FUNCTION_BLOCK FB_Janitza
VAR_IN_OUT
	get					: ST_PowerMonitor_get;
	b_ThirdOutputFieldAvailable	: BOOL;
	b_NeutralTransformerAvailable: BOOL;
	b_InputFieldsAvailable		: BOOL;
END_VAR
VAR
	MBRead: FB_MBReadRegs;
	t_MBTimeout				: 	TIME := T#500MS;
	w_MBStartAddress		:	WORD;
	//Set 1 is bigger, as this includes voltage measurements.
	DataBuffer				: 	ARRAY[0..62] OF REAL;
	//SecondDataBuffer		: 	ARRAY[0..62] OF REAL;
	UI_Iterator	:	UINT;
	//retrieve new data every 100ms
	GetDataTimer	:	TON := (PT := TIME#50MS);
	
	di_RotationState		: DINT;
	
	ton_DelaySFCTip			: TON := (PT := T#10MS);
	
	
END_VAR

VAR_INPUT
	ReadData: BOOL;
	b_TNmodeEnable		AT %Q* : BOOL;
	
END_VAR

VAR
	ast_InputPowerlockData	:	ARRAY[1..2] OF ST_MeasurementFieldData;
	ast_OutputPowerlockData	:	ARRAY[1..3] OF ST_MeasurementFieldData;

	StartTransmissionEdge : R_Trig;
	TransmissionDone	:	F_trig;
	
	ui_MBRetryCount	:	uint;
	
	b_busy: BOOL;
	b_CommError: BOOL;
	udi_errid: UDINT;
	udi_cbread: UDINT;
	
END_VAR

//Initialization
get.events.b_MBCommWarning := FALSE;
get.events.b_MBCommError := FALSE;

MBread(tTimeOut := t_MBTimeout);

//While ReadData is true, initiate data transfer every 100ms;
GetDataTimer(in:= ((NOT GetDataTimer.Q) AND ReadData));

//ReadJanitzaData();
ReadDataSFC();

ACTION aCombineInputData:
IF b_InputFieldsAvailable THEN
	//Combine shared data from output fields into get struct
	get.InputField.ar_Current[Phases.L1] :=	get.InputField.powerlock[1].ar_Current[Phases.L1] + 
											get.InputField.Powerlock[2].ar_Current[Phases.L1];
	
	get.InputField.ar_Current[Phases.L2] :=	get.InputField.powerlock[1].ar_Current[Phases.L2] + 
											get.InputField.powerlock[2].ar_Current[Phases.L2];
	
	get.InputField.ar_Current[Phases.L3] :=	get.InputField.powerlock[1].ar_Current[Phases.L3] + 
											get.InputField.powerlock[2].ar_Current[Phases.L3];			
	
	get.InputField.ar_Current[Phases.N] :=	get.InputField.powerlock[1].ar_Current[Phases.N] + 
											get.InputField.powerlock[2].ar_Current[Phases.N];			
	
	get.InputField.ar_Current[Phases.AVG] :=	(get.InputField.ar_Current[Phases.L1] + 
											get.InputField.ar_Current[Phases.L2] +
											get.InputField.ar_Current[Phases.L3])/3;							
	
	Get.InputField.ar_ActivePower[Phases.L1]	:=	get.InputField.powerlock[1].ar_ActivePower[Phases.L1] + get.InputField.powerlock[2].ar_ActivePower[Phases.L1];
	Get.InputField.ar_ActivePower[Phases.L2]	:=	get.InputField.powerlock[1].ar_ActivePower[Phases.L2] + get.InputField.powerlock[2].ar_ActivePower[Phases.L2];
	Get.InputField.ar_ActivePower[Phases.L3]	:=	get.InputField.powerlock[1].ar_ActivePower[Phases.L3] + get.InputField.powerlock[2].ar_ActivePower[Phases.L3];
	Get.InputField.ar_ActivePower[Phases.AVG]	:=	get.InputField.powerlock[1].ar_ActivePower[Phases.AVG] + get.InputField.powerlock[2].ar_ActivePower[Phases.AVG];									
	Get.InputField.ar_ApparentPower[Phases.L1]	:=	get.InputField.powerlock[1].ar_ApparentPower[Phases.L1] + get.InputField.powerlock[2].ar_ApparentPower[Phases.L1];
	Get.InputField.ar_ApparentPower[Phases.L2]	:=	get.InputField.powerlock[1].ar_ApparentPower[Phases.L2] + get.InputField.powerlock[2].ar_ApparentPower[Phases.L2];	
	Get.InputField.ar_ApparentPower[Phases.L3]	:=	get.InputField.powerlock[1].ar_ApparentPower[Phases.L3] + get.InputField.powerlock[2].ar_ApparentPower[Phases.L3];
	Get.InputField.ar_ApparentPower[Phases.AVG]	:=	get.InputField.powerlock[1].ar_ApparentPower[Phases.AVG] + get.InputField.powerlock[2].ar_ApparentPower[Phases.AVG];												
	Get.InputField.ar_ReactivePower[Phases.L1]	:=	get.InputField.powerlock[1].ar_ReactivePower[Phases.L1] + get.InputField.powerlock[2].ar_ReactivePower[Phases.L1];
	Get.InputField.ar_ReactivePower[Phases.L2]	:=	get.InputField.powerlock[1].ar_ReactivePower[Phases.L2] + get.InputField.powerlock[2].ar_ReactivePower[Phases.L2];											
	Get.InputField.ar_ReactivePower[Phases.L3]	:=	get.InputField.powerlock[1].ar_ReactivePower[Phases.L3] + get.InputField.powerlock[2].ar_ReactivePower[Phases.L3];								
	Get.InputField.ar_ReactivePower[Phases.AVG]	:=	get.InputField.powerlock[1].ar_ReactivePower[Phases.AVG] + get.InputField.powerlock[2].ar_ReactivePower[Phases.AVG];	

	Get.InputField.r_EnergyConsumed		:=	get.InputField.powerlock[1].r_EnergyConsumed + 
											get.InputField.powerlock[2].r_EnergyConsumed;
	
	Get.InputField.r_EnergySupplied		:=	get.InputField.powerlock[1].r_EnergySupplied + 
											get.InputField.powerlock[2].r_EnergySupplied;
	
	get.InputField.ar_PowerFactor[Phases.L1] 	:=  PowerFactor(Get.InputField.ar_activePower[Phases.L1], Get.InputField.ar_ApparentPower[Phases.L1], Get.InputField.ar_ReactivePower[Phases.L1]); 										
	get.InputField.ar_PowerFactor[Phases.L2] 	:=  PowerFactor(Get.InputField.ar_activePower[Phases.L2], Get.InputField.ar_ApparentPower[Phases.L2], Get.InputField.ar_ReactivePower[Phases.L2]); 		
	get.InputField.ar_PowerFactor[Phases.L3] 	:=  PowerFactor(Get.InputField.ar_activePower[Phases.L3], Get.InputField.ar_ApparentPower[Phases.L3], Get.InputField.ar_ReactivePower[Phases.L3]); 									
	get.InputField.ar_THD[Phases.L1] 		:=		(ast_InputPowerLockData[1].ar_THD[Phases.L1] + ast_InputPowerLockData[2].ar_THD[Phases.L1])/2;		
	get.InputField.ar_THD[Phases.L2] 		:=		(ast_InputPowerLockData[1].ar_THD[Phases.L2] + ast_InputPowerLockData[2].ar_THD[Phases.L2])/2;	
	get.InputField.ar_THD[Phases.L3]		:=		(ast_InputPowerLockData[1].ar_THD[Phases.L3] + ast_InputPowerLockData[2].ar_THD[Phases.L3])/2;											
	get.InputField.ar_PowerFactor[Phases.AVG] :=	(get.InputField.ar_PowerFactor[Phases.L1] + get.InputField.ar_PowerFactor[Phases.L2] + get.InputField.ar_PowerFactor[Phases.L3])/3;		
	get.InputField.ar_THD[Phases.AVG] :=			(get.InputField.ar_THD[Phases.L1] + get.InputField.ar_THD[Phases.L2] + get.InputField.ar_THD[Phases.L3])/3;
END_IF
END_ACTION

ACTION aCombineOutputData:
//Combine shared data from output fields into get struct
get.OutputField.ar_Current[Phases.L1] 	:=	get.OutputField.powerlock[1].ar_current[Phases.L1] + get.OutputField.powerlock[2].ar_current[Phases.L1] + get.OutputField.powerlock[3].ar_current[Phases.L1];
get.OutputField.ar_Current[Phases.L2] 	:=	get.OutputField.powerlock[1].ar_current[Phases.L2] + get.OutputField.powerlock[2].ar_current[Phases.L2] + get.OutputField.powerlock[3].ar_current[Phases.L2];
get.OutputField.ar_Current[Phases.L3] 	:=	get.OutputField.powerlock[1].ar_current[Phases.L3] + get.OutputField.powerlock[2].ar_current[Phases.L3] + get.OutputField.powerlock[3].ar_current[Phases.L3];			
get.OutputField.ar_Current[Phases.N] 	:=	get.OutputField.powerlock[1].ar_current[Phases.N] + get.OutputField.powerlock[2].ar_current[Phases.N] + get.OutputField.powerlock[3].ar_current[Phases.N];			
get.OutputField.ar_Current[Phases.AVG] :=	(get.OutputField.ar_Current[Phases.L1] + get.OutputField.ar_Current[Phases.L2] + get.OutputField.ar_Current[Phases.L3])/3;							

Get.OutputField.ar_ActivePower[Phases.L1]		:=	get.outputfield.powerlock[1].ar_ActivePower[Phases.L1] + 
													get.outputfield.powerlock[2].ar_ActivePower[Phases.L1] +
													get.outputfield.powerlock[3].ar_ActivePower[Phases.L1];
Get.OutputField.ar_ActivePower[Phases.L2]		:=	get.outputfield.powerlock[1].ar_ActivePower[Phases.L2] + 
													get.outputfield.powerlock[2].ar_ActivePower[Phases.L2] +
													get.outputfield.powerlock[3].ar_ActivePower[Phases.L2];				
Get.OutputField.ar_ActivePower[Phases.L3]		:=	get.outputfield.powerlock[1].ar_ActivePower[Phases.L3] + 
													get.outputfield.powerlock[2].ar_ActivePower[Phases.L3] + 
													get.outputfield.powerlock[3].ar_ActivePower[Phases.L3];												
Get.OutputField.ar_ActivePower[Phases.AVG]		:=	get.outputfield.powerlock[1].ar_ActivePower[Phases.AVG] + 
													get.outputfield.powerlock[2].ar_ActivePower[Phases.AVG] +
													get.outputfield.powerlock[3].ar_ActivePower[Phases.AVG];																				
Get.OutputField.ar_ApparentPower[Phases.L1]		:=	get.outputfield.powerlock[1].ar_ApparentPower[Phases.L1] + 
													get.outputfield.powerlock[2].ar_ApparentPower[Phases.L1] +
													get.outputfield.powerlock[3].ar_ApparentPower[Phases.L1];
Get.OutputField.ar_ApparentPower[Phases.L2]		:=	get.outputfield.powerlock[1].ar_ApparentPower[Phases.L2] + 
													get.outputfield.powerlock[2].ar_ApparentPower[Phases.L2] +
													get.outputfield.powerlock[3].ar_ApparentPower[Phases.L2];													
Get.OutputField.ar_ApparentPower[Phases.L3]		:=	get.outputfield.powerlock[1].ar_ApparentPower[Phases.L3] + 
													get.outputfield.powerlock[2].ar_ApparentPower[Phases.L3] +
													get.outputfield.powerlock[3].ar_ApparentPower[Phases.L3];													
Get.OutputField.ar_ApparentPower[Phases.AVG]	:=	get.outputfield.powerlock[1].ar_ApparentPower[Phases.AVG] + 
													get.outputfield.powerlock[2].ar_ApparentPower[Phases.AVG] +
													get.outputfield.powerlock[3].ar_ApparentPower[Phases.AVG];																																								
Get.OutputField.ar_ReactivePower[Phases.L1]		:=	get.outputfield.powerlock[1].ar_ReactivePower[Phases.L1] + 
													get.outputfield.powerlock[2].ar_ReactivePower[Phases.L1] +
													get.outputfield.powerlock[3].ar_ReactivePower[Phases.L1];		
Get.OutputField.ar_ReactivePower[Phases.L2]		:=	get.outputfield.powerlock[1].ar_ReactivePower[Phases.L2] + 
													get.outputfield.powerlock[2].ar_ReactivePower[Phases.L2] +
													get.outputfield.powerlock[3].ar_ReactivePower[Phases.L2];															
Get.OutputField.ar_ReactivePower[Phases.L3]		:=	get.outputfield.powerlock[1].ar_ReactivePower[Phases.L3] + 
													get.outputfield.powerlock[2].ar_ReactivePower[Phases.L3] +
													get.outputfield.powerlock[3].ar_ReactivePower[Phases.L3];															
Get.OutputField.ar_ReactivePower[Phases.AVG]	:=	get.outputfield.powerlock[1].ar_ReactivePower[Phases.AVG] + 
													get.outputfield.powerlock[2].ar_ReactivePower[Phases.AVG] +	
													get.outputfield.powerlock[3].ar_ReactivePower[Phases.AVG];																					
Get.OutputField.r_EnergyConsumed				:=	get.outputfield.powerlock[1].r_EnergyConsumed + 
													get.outputfield.powerlock[2].r_EnergyConsumed + 
													get.outputfield.powerlock[3].r_EnergyConsumed;
Get.OutputField.r_EnergySupplied				:=	get.outputfield.powerlock[1].r_EnergySupplied + 
													get.outputfield.powerlock[2].r_EnergySupplied + 
													get.outputfield.powerlock[3].r_EnergySupplied;
get.OutputField.ar_PowerFactor[Phases.L1] 		:=  PowerFactor(Get.OutputField.ar_activePower[Phases.L1], Get.OutputField.ar_ApparentPower[Phases.L1], Get.OutputField.ar_ReactivePower[Phases.L1]); 										
get.OutputField.ar_PowerFactor[Phases.L2] 		:=  PowerFactor(Get.OutputField.ar_activePower[Phases.L2], Get.OutputField.ar_ApparentPower[Phases.L2], Get.OutputField.ar_ReactivePower[Phases.L2]); 		
get.OutputField.ar_PowerFactor[Phases.L3] 		:=  PowerFactor(Get.OutputField.ar_activePower[Phases.L3], Get.OutputField.ar_ApparentPower[Phases.L3], Get.OutputField.ar_ReactivePower[Phases.L3]); 									

//if 3 output fields are available, calculate averages over 3 fields. Otherwise over 2
IF b_ThirdOutputFieldAvailable THEN
	get.OutputField.ar_THD[Phases.L1] 		:=	   (get.outputfield.powerlock[1].ar_THD[Phases.L1] + 
													get.outputfield.powerlock[2].ar_THD[Phases.L1] + 
													get.outputfield.powerlock[3].ar_THD[Phases.L1])/3;												
	get.OutputField.ar_THD[Phases.L2] 		:=     (get.outputfield.powerlock[1].ar_THD[Phases.L2] + 
													get.outputfield.powerlock[2].ar_THD[Phases.L2] + 
													get.outputfield.powerlock[3].ar_THD[Phases.L2])/3;		
	get.OutputField.ar_THD[Phases.L3]		 :=	   (get.outputfield.powerlock[1].ar_THD[Phases.L3] + 
													get.outputfield.powerlock[2].ar_THD[Phases.L3] + 
													get.outputfield.powerlock[3].ar_THD[Phases.L3])/3;														
ELSE
	get.OutputField.ar_THD[Phases.L1] 		:=	   (get.outputfield.powerlock[1].ar_THD[Phases.L1] + 
													get.outputfield.powerlock[2].ar_THD[Phases.L1])/2;											
	get.OutputField.ar_THD[Phases.L2] 		:=     (get.outputfield.powerlock[1].ar_THD[Phases.L2] + 
													get.outputfield.powerlock[2].ar_THD[Phases.L2])/2;	
	get.OutputField.ar_THD[Phases.L3]		 :=	   (get.outputfield.powerlock[1].ar_THD[Phases.L3] + 
													get.outputfield.powerlock[2].ar_THD[Phases.L3])/2;											
END_IF



get.OutputField.ar_PowerFactor[Phases.AVG] :=	(get.OutputField.ar_PowerFactor[Phases.L1] + 
												get.OutputField.ar_PowerFactor[Phases.L2] + 
												get.OutputField.ar_PowerFactor[Phases.L3])/3;		

get.OutputField.ar_THD[Phases.AVG] :=			(get.OutputField.ar_THD[Phases.L1] + 
												get.OutputField.ar_THD[Phases.L2] + 
												get.OutputField.ar_THD[Phases.L3])/3;
												
get.OutputField.r_VoltageUnbalance := 			LineUnbalance(
													r_L1 := get.OutputField.ar_LineVoltage[phases.L1],
													r_L2 := get.OutputField.ar_LineVoltage[phases.L2],
													r_L3 := get.OutputField.ar_LineVoltage[phases.L3]);
													
get.OutputField.r_CurrentUnbalance := 			LineUnbalance(
													r_L1 := get.OutputField.ar_Current[phases.L1], 
													r_L2 := get.OutputField.ar_Current[phases.L2], 
													r_L3 := get.OutputField.ar_Current[phases.L3]);
END_ACTION

ACTION aReadInputField1:
IF NOT b_InputFieldsAvailable THEN
	//skip this step if input fields are not in use
	ton_DelaySFCTip(IN:= TRUE);
	SFCTip := ton_DelaySFCTip.Q;
ELSE
	
//	IF b_ThirdOutputFieldAvailable THEN
//		//if third output field is available, Input field 1 is connected to module 2, so inputfield 1 is address 19600
//		w_MBStartAddress := 19600;
//	ELSE
//		//if no third output field is available, Input field 1 is connected to module 1, so inputfield 1 is address 19400
//		w_MBStartAddress := 19400;
//	END_IF

	MBRead(
	sIPAddr := PowerMeterConfig.IP_JANITZA,
	nTCPPort := PowerMeterConfig.MBPort_Janitza,
	nUnitID := 1,//16#FF;
	nMBAddr := 19600,//w_MBStartAddress,
	nQuantity := 50*2,
	cbLength := SIZEOF(DataBuffer),
	pDestAddr := ADR(DataBuffer),
	bExecute := NOT (b_busy OR TransmissionDone.Q),	//	<- werkt dit niet gewoon?
	bBusy => b_busy,
	bError => b_CommError,
	nErrId => udi_errid,
	cbRead => udi_cbread,
	);
	
	TransmissionDone(clk := b_busy);
	
	IF TransmissionDone.q THEN
		IF NOT b_CommError  THEN
			MapMeasuringField(firstfield := False, buffer := databuffer, data := get.InputField.Powerlock[1]);		
			ui_MBRetryCount := 0;
			sfctip := TRUE;
		ELSE
			ui_MBRetryCount := ui_MBRetryCount + 1;
			
			IF ui_MBRetryCount > 1 THEN
				get.events.b_MBCommWarning := TRUE;
			END_IF	
			
			//if comm fails 5 times in a row. try next input
			IF ui_MBRetryCount > 4 THEN
				get.Events.b_MBCommError := TRUE;
				ton_DelaySFCTip(IN:= TRUE);
				SFCTip := ton_DelaySFCTip.Q;
			END_IF
		END_IF
	END_IF
END_IF

IF MBRead.bError THEN
	MBRead.bError;
END_IF
END_ACTION

ACTION aReadInputField2:
IF NOT b_InputFieldsAvailable THEN
	//skip this step if input fields are not in use
	ton_DelaySFCTip(IN:= TRUE);
	SFCTip := ton_DelaySFCTip.Q;
ELSE
	
//	IF b_ThirdOutputFieldAvailable THEN
//		//if third output field is available, Input field is connected to bottom of module 2, so inputfield 2 is address 19700
//		w_MBStartAddress := 19700;
//	ELSE
//		//if no third output field is available, Input field is connected to top of module 1, so inputfield 2 is address 19500
//		w_MBStartAddress := 19600;
//	END_IF

	MBRead(
	sIPAddr := PowerMeterConfig.IP_JANITZA,
	nTCPPort := PowerMeterConfig.MBPort_Janitza,
	nUnitID := 1,//16#FF;
	nMBAddr := 19700,//w_MBStartAddress,
	nQuantity := 50*2,
	cbLength := SIZEOF(DataBuffer),
	pDestAddr := ADR(DataBuffer),
	bExecute := NOT (b_busy OR TransmissionDone.Q),	//	<- werkt dit niet gewoon?
	bBusy => b_busy,
	bError => b_CommError,
	nErrId => udi_errid,
	cbRead => udi_cbread,
	);
	
	TransmissionDone(clk := b_busy);
	
	IF TransmissionDone.q THEN
		IF NOT b_CommError THEN	
			MapMeasuringField(firstfield := False, buffer := databuffer, data := get.InputField.Powerlock[2]);
			ui_MBRetryCount := 0;
			sfctip := TRUE;
		ELSE
			ui_MBRetryCount := ui_MBRetryCount + 1;
			
			
			IF ui_MBRetryCount > 1 THEN
				get.events.b_MBCommWarning := TRUE;
			END_IF	
			
			//if comm fails 5 times in a row. try next input
			IF ui_MBRetryCount > 4 THEN
				get.Events.b_MBCommError := TRUE;
				ton_DelaySFCTip(IN:= TRUE);
				SFCTip := ton_DelaySFCTip.Q;
			END_IF
		END_IF
	END_IF
END_IF
END_ACTION

ACTION aReadInternalField:
MBRead(
sIPAddr := PowerMeterConfig.IP_JANITZA,
nTCPPort := PowerMeterConfig.MBPort_Janitza,
nUnitID := 1,//16#FF;
nMBAddr := 19300,
nQuantity := 50*2,
cbLength := SIZEOF(DataBuffer),
pDestAddr := ADR(DataBuffer),
bExecute := NOT (b_busy OR TransmissionDone.Q),	//	<- werkt dit niet gewoon?
bBusy => b_busy,
bError => b_CommError,
nErrId => udi_errid,
cbRead => udi_cbread,
);

TransmissionDone(clk := b_busy);

IF TransmissionDone.q THEN
	IF NOT b_CommError  THEN
			MapMeasuringField(firstfield := False, buffer := databuffer, data := get.InternalSupply);
		ui_MBRetryCount := 0;
		sfctip := TRUE;
	ELSE
		ui_MBRetryCount := ui_MBRetryCount + 1;
				
		IF ui_MBRetryCount > 1 THEN
			get.events.b_MBCommWarning := TRUE;
		END_IF	
		
		//if comm fails 5 times in a row. try next input
		IF ui_MBRetryCount > 4 THEN
			get.Events.b_MBCommError := TRUE;
			ton_DelaySFCTip(IN:= TRUE);
			SFCTip := ton_DelaySFCTip.Q;
		END_IF
	END_IF
END_IF
END_ACTION

ACTION aReadNeutralBess:

IF NOT b_NeutraltransformerAvailable THEN
	//skip this step if third field isn't in use
	ton_DelaySFCTip(IN:= TRUE);
	SFCTip := ton_DelaySFCTip.Q;
ELSE
	MBRead(
	sIPAddr := PowerMeterConfig.IP_JANITZA,
	nTCPPort := PowerMeterConfig.MBPort_Janitza,
	nUnitID := 1,//16#FF;
	nMBAddr := 19500,
	nQuantity := 4*2,
	cbLength := SIZEOF(DataBuffer), //second databuffer replaced
	pDestAddr := ADR(DataBuffer),
	bExecute := NOT (b_busy OR TransmissionDone.Q),	//	<- werkt dit niet gewoon?
	bBusy => b_busy,
	bError => b_CommError,
	nErrId => udi_errid,
	cbRead => udi_cbread,
	);
	
	TransmissionDone(clk := b_busy);
	
	IF TransmissionDone.q THEN
		IF NOT b_CommError  THEN	
		
			//field specific data, keep separate at first. Then combine data into get struct in a later step.
			ChangeRealEndianess(IN := Databuffer[3], 1.0, get.BESS.ar_Current[Phases.N]);
			ui_MBRetryCount := 0;
			sfctip := TRUE;
		ELSE
			ui_MBRetryCount := ui_MBRetryCount + 1;

			IF ui_MBRetryCount > 1 THEN
				get.events.b_MBCommWarning := TRUE;
			END_IF	
			
			//if comm fails 5 times in a row. try next input
			IF ui_MBRetryCount > 4 THEN
				get.Events.b_MBCommError := TRUE;
				ton_DelaySFCTip(IN:= TRUE);
				SFCTip := ton_DelaySFCTip.Q;
			END_IF
		END_IF
	END_IF
END_IF
END_ACTION

ACTION aReadOutputField1:
get.events.b_ACdirectionDataInvalid := FALSE;

MBRead(
sIPAddr := PowerMeterConfig.IP_JANITZA,
nTCPPort := PowerMeterConfig.MBPort_Janitza,
nUnitID := 1,
nMBAddr := 19000,
nQuantity := 61*2,
cbLength := SIZEOF(DataBuffer),
pDestAddr := ADR(DataBuffer),
bExecute := NOT (b_busy OR TransmissionDone.Q),	//	<- werkt dit niet gewoon?
bBusy => b_busy,
bError => b_CommError,
nErrId => udi_errid,
cbRead => udi_cbread,
);

TransmissionDone(clk := b_busy);

IF TransmissionDone.q THEN
	IF NOT b_CommError THEN
		
		Mapvoltagefield(buffer := databuffer, data := get.OutputField);
		MapMeasuringField(firstfield := True, buffer := databuffer, data := get.OutputField.Powerlock[1]);
		ui_MBRetryCount := 0;
		sfctip := TRUE;
	ELSE
		ui_MBRetryCount := ui_MBRetryCount + 1;
		
		IF ui_MBRetryCount > 1 THEN
			get.events.b_MBCommWarning := TRUE;
		END_IF	
		
		//if comm fails 5 times in a row. try next input
		IF ui_MBRetryCount > 4 THEN
			get.Events.b_MBCommError := TRUE;
			ton_DelaySFCTip(IN:= TRUE);
			SFCTip := ton_DelaySFCTip.Q;
		END_IF
	END_IF
END_IF
END_ACTION

ACTION aReadOutputField2:
MBRead(
sIPAddr := PowerMeterConfig.IP_JANITZA,
nTCPPort := PowerMeterConfig.MBPort_Janitza,
nUnitID := 1,//16#FF,
nMBAddr := 19200,
nQuantity := 50*2,
cbLength := SIZEOF(DataBuffer),
pDestAddr := ADR(DataBuffer),
bExecute := NOT (b_busy OR TransmissionDone.Q),	//	<- werkt dit niet gewoon?
bBusy => b_busy,
bError => b_CommError,
nErrId => udi_errid,
cbRead => udi_cbread,
);

TransmissionDone(clk := b_busy);

IF TransmissionDone.q THEN
	IF NOT b_CommError THEN	
		MapMeasuringField(firstfield := False, buffer := databuffer, data := get.OutputField.Powerlock[2]);
		ui_MBRetryCount := 0;
		sfctip := TRUE;
	ELSE
		ui_MBRetryCount := ui_MBRetryCount + 1;
		
		IF ui_MBRetryCount > 1 THEN
			get.events.b_MBCommWarning := TRUE;
		END_IF	
		
		//if comm fails 5 times in a row. try next input
		IF ui_MBRetryCount > 4 THEN
			get.Events.b_MBCommError := TRUE;
			ton_DelaySFCTip(IN:= TRUE);
			SFCTip := ton_DelaySFCTip.Q;
		END_IF
	END_IF
END_IF
END_ACTION

ACTION aReadOutputField3:
IF NOT b_ThirdOutputFieldAvailable THEN
	//skip this step if third field isn't in use
	ton_DelaySFCTip(IN:= TRUE);
	SFCTip := ton_DelaySFCTip.Q;
ELSE
	MBRead(
	sIPAddr := PowerMeterConfig.IP_JANITZA,
	nTCPPort := PowerMeterConfig.MBPort_Janitza,
	nUnitID := 1,//16#FF;
	nMBAddr := 19400,
	nQuantity := 50*2,
	cbLength := SIZEOF(DataBuffer), //second databuffer replaced
	pDestAddr := ADR(DataBuffer),
	bExecute := NOT (b_busy OR TransmissionDone.Q),	//	<- werkt dit niet gewoon?
	bBusy => b_busy,
	bError => b_CommError,
	nErrId => udi_errid,
	cbRead => udi_cbread,
	);
	
	TransmissionDone(clk := b_busy);
	
	IF TransmissionDone.q THEN
		IF NOT b_CommError  THEN
			MapMeasuringField(firstfield := False, buffer := databuffer, data := get.OutputField.Powerlock[3]);	
			ui_MBRetryCount := 0;
			sfctip := TRUE;
		ELSE
			ui_MBRetryCount := ui_MBRetryCount + 1;

			IF ui_MBRetryCount > 1 THEN
				get.events.b_MBCommWarning := TRUE;
			END_IF	
			
			//if comm fails 5 times in a row. try next input
			IF ui_MBRetryCount > 4 THEN
				get.Events.b_MBCommError := TRUE;
				ton_DelaySFCTip(IN:= TRUE);
				SFCTip := ton_DelaySFCTip.Q;
			END_IF
		END_IF
	END_IF
END_IF
END_ACTION

METHOD ChangeRealEndianess
VAR_INPUT
	IN				: REAL;
	scale			: REAL;
END_VAR

VAR_IN_OUT
	variable 		: REAL;
END_VAR

VAR_INST
	tempreal		: REAL;
	tempdword		: DWORD;
	testword		: WORD;	
END_VAR
//tempdword := PDWORD_TO_DWORD(ADR(InputReal));
//memcpy(ADR(TestWord), ADR(tempdword), 2);
//tempdword := ROL(tempdword, 16);

tempdword := PDWORD_TO_DWORD(ADR(IN));
tempdword := ROL(tempdword, 16);
tempreal := PREAL_TO_REAL(ADR(tempdword));

IF NOT IsNaN(tempreal) THEN
	variable := tempreal * scale;
END_IF
END_METHOD

METHOD MapMeasuringField
VAR_INPUT
	FirstField		: BOOL;
END_VAR
VAR_IN_OUT
	buffer 		: ARRAY[*] OF REAL;
	data 		: ST_MeasurementFieldData;
END_VAR

VAR_INST
	iterStartIndex 	: WORD;
	iterator	: WORD;
	tempreal	: REAL;
END_VAR
iterStartIndex := SEL(firstfield, 0, 6);

FOR iterator := 0 TO 20 DO
	tempreal := Buffer[iterator + iterstartindex];
	CASE iterator OF
		0: ChangeRealEndianess(tempreal, 1, data.ar_Current[Phases.L1]);
		1: ChangeRealEndianess(tempreal, 1, data.ar_Current[Phases.L2]);
		2: ChangeRealEndianess(tempreal, 1, data.ar_Current[Phases.L3]);
		3: ChangeRealEndianess(tempreal, 1, data.ar_Current[Phases.N]);
		4: ChangeRealEndianess(tempreal, 0.001, data.ar_ActivePower[phases.L1]);
		5: ChangeRealEndianess(tempreal, 0.001, data.ar_ActivePower[phases.L2]);
		6: ChangeRealEndianess(tempreal, 0.001, data.ar_ActivePower[phases.L3]);
		7: ChangeRealEndianess(tempreal, 0.001, data.ar_ActivePower[phases.AVG]);
		8: ChangeRealEndianess(tempreal, 0.001, data.ar_ApparentPower[phases.L1]);
		9: ChangeRealEndianess(tempreal, 0.001, data.ar_ApparentPower[phases.L2]);
		10: ChangeRealEndianess(tempreal, 0.001, data.ar_ApparentPower[phases.L3]);
		11: ChangeRealEndianess(tempreal, 0.001, data.ar_ApparentPower[phases.AVG]);
		12: ChangeRealEndianess(tempreal, 0.001, data.ar_ReactivePower[phases.L1]);
		13: ChangeRealEndianess(tempreal, 0.001, data.ar_ReactivePower[phases.L2]);
		14: ChangeRealEndianess(tempreal, 0.001, data.ar_ReactivePower[phases.L3]);
		15:	ChangeRealEndianess(tempreal, 0.001, data.ar_ReactivePower[phases.AVG]);
		16: ChangeRealEndianess(tempreal, 1, data.ar_powerfactor[phases.L1]);
		17: ChangeRealEndianess(tempreal, 1, data.ar_powerfactor[phases.L2]);
		18: ChangeRealEndianess(tempreal, 1, data.ar_powerfactor[phases.L3]);
		
	END_CASE
END_FOR 

IF firstfield THEN
	ChangeRealEndianess(buffer[34], 0.001, data.r_EnergySupplied);
	ChangeRealEndianess(buffer[38], 0.001, data.r_EnergyConsumed);
	ChangeRealEndianess(buffer[58], 1, data.ar_THD[Phases.L1]);
	ChangeRealEndianess(buffer[59], 1, data.ar_THD[Phases.L2]);
	ChangeRealEndianess(buffer[60], 1, data.ar_THD[Phases.L3]);
ELSE
	ChangeRealEndianess(buffer[26], 0.001, data.r_EnergySupplied);
	ChangeRealEndianess(buffer[30], 0.001, data.r_EnergyConsumed);
	ChangeRealEndianess(buffer[47], 1, data.ar_THD[Phases.L1]);
	ChangeRealEndianess(buffer[48], 1, data.ar_THD[Phases.L2]);
	ChangeRealEndianess(buffer[49], 1, data.ar_THD[Phases.L3]);
END_IF




data.ar_Current[Phases.AVG] := (data.ar_Current[Phases.L1] + data.ar_Current[Phases.L2] + data.ar_Current[Phases.L3])/3;
data.ar_powerfactor[phases.AVG] := (data.ar_powerfactor[phases.L1] + data.ar_powerfactor[phases.L2] + data.ar_powerfactor[phases.L3])/3;
data.ar_THD[phases.AVG] := (data.ar_THD[phases.L1] + data.ar_THD[phases.L2] + data.ar_THD[phases.L3])/3;
data.r_CurrentUnbalance := LineUnbalance(r_L1 := data.ar_Current[Phases.L1], r_L2 := data.ar_Current[Phases.L1], r_L3 :=  data.ar_Current[Phases.L3]);
END_METHOD

METHOD MapVoltageField

VAR_IN_OUT
	buffer 			: 	ARRAY[*] OF REAL;
	data			: ST_measurementVoltageData;
END_VAR

VAR
	i_rotation : INT;
END_VAR

VAR
	iterator	: WORD;
	tempreal	: REAL;
END_VAR
FOR iterator := 0 TO 7 DO
	tempreal := Buffer[iterator];
	CASE iterator OF
		0: ChangeRealEndianess(tempreal,1, data.ar_PhaseVoltage[Phases.L1]);
		1: ChangeRealEndianess(tempreal,1, data.ar_PhaseVoltage[Phases.L2]);
		2: ChangeRealEndianess(tempreal,1, data.ar_PhaseVoltage[Phases.L3]);
		3: ChangeRealEndianess(tempreal,1, data.ar_LineVoltage[Phases.L1]);
		4: ChangeRealEndianess(tempreal,1, data.ar_LineVoltage[Phases.L2]);
		5: ChangeRealEndianess(tempreal,1, data.ar_LineVoltage[Phases.L3]);
	END_CASE
END_FOR 

MEMCPY(ADR(i_rotation), ADR(Buffer[26])+2, 2);
CASE i_rotation OF
	-1 	:	data.e_ACrotationStatus := eACRotationState.Left;
	1	:	data.e_ACrotationStatus := eACRotationState.Right;
	0	:	data.e_ACrotationStatus := eACRotationState.None;
	ELSE
		get.events.b_ACdirectionDataInvalid := TRUE;
END_CASE

ChangeRealEndianess(Buffer[19], 1, data.ar_Frequency[0]);

IF data.ar_LineVoltage[Phases.AVG] < 360 THEN
	data.e_ACrotationStatus := eACRotationState.None;
END_IF

data.ar_PhaseVoltage[0] := (data.ar_PhaseVoltage[Phases.L1] + data.ar_PhaseVoltage[Phases.L2] + data.ar_PhaseVoltage[Phases.L3]) / 3;
data.ar_LineVoltage[0] := (data.ar_LineVoltage[Phases.L1] + data.ar_LineVoltage[Phases.L2] + data.ar_LineVoltage[Phases.L3]) / 3;
data.r_VoltageUnbalance := LineUnbalance(r_L1 := data.ar_LineVoltage[Phases.L1], r_L2 := data.ar_LineVoltage[Phases.L2], r_L3 :=  data.ar_LineVoltage[Phases.L3]);
END_METHOD

ACTION ReadDataSFC:
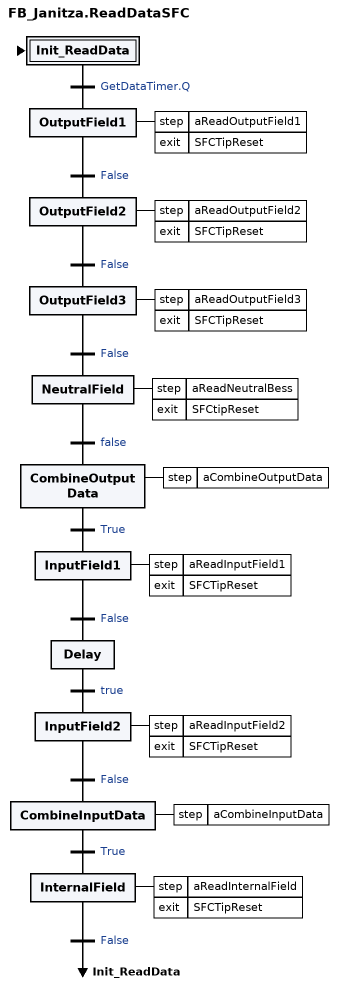
INITIAL_STEP Init_ReadData:
END_STEP
TRANSITION FROM Init_ReadData TO OutputField1
    := GetDataTimer.Q;
END_TRANSITION
STEP OutputField1:
    aReadOutputField1(N);  // step action
    SFCTipReset(P0);  // exit action
END_STEP
TRANSITION FROM OutputField1 TO OutputField2
    := False;
END_TRANSITION
STEP OutputField2:
    aReadOutputField2(N);  // step action
    SFCTipReset(P0);  // exit action
END_STEP
TRANSITION FROM OutputField2 TO OutputField3
    := False;
END_TRANSITION
STEP OutputField3:
    aReadOutputField3(N);  // step action
    SFCTipReset(P0);  // exit action
END_STEP
TRANSITION FROM OutputField3 TO NeutralField
    := False;
END_TRANSITION
STEP NeutralField:
    aReadNeutralBess(N);  // step action
    SFCtipReset(P0);  // exit action
END_STEP
TRANSITION FROM NeutralField TO CombineOutputData
    := false;
END_TRANSITION
STEP CombineOutputData:
    aCombineOutputData(N);  // step action
END_STEP
TRANSITION FROM CombineOutputData TO InputField1
    := True;
END_TRANSITION
STEP InputField1:
    aReadInputField1(N);  // step action
    SFCTipReset(P0);  // exit action
END_STEP
TRANSITION FROM InputField1 TO Delay
    := False;
END_TRANSITION
STEP Delay:  // min time T#10ms
END_STEP
TRANSITION FROM Delay TO InputField2
    := true;
END_TRANSITION
STEP InputField2:
    aReadInputField2(N);  // step action
    SFCTipReset(P0);  // exit action
END_STEP
TRANSITION FROM InputField2 TO CombineInputData
    := False;
END_TRANSITION
STEP CombineInputData:
    aCombineInputData(N);  // step action
END_STEP
TRANSITION FROM CombineInputData TO InternalField
    := True;
END_TRANSITION
STEP InternalField:
    aReadInternalField(N);  // step action
    SFCTipReset(P0);  // exit action
END_STEP
TRANSITION FROM InternalField TO Init_ReadData
    := False;
END_TRANSITION
END_ACTION

ACTION SFCTipReset:
ton_DelaySFCTip(IN:= FALSE);
SFCTip := ton_DelaySFCTip.Q;
END_ACTION

END_FUNCTION_BLOCK

(* stored: Version 1.1.0.1, ProductVersion 3.1.4024.12
   POU FB_Janitza: Id {39a3b041-a991-4c24-856c-d797ef0b9fe6}, SpecialFunc None
   Folder SFC: Id {7b546ac8-05b5-4879-b9ec-fda86df5f1f4}
   Action aCombineInputData: Id {180e600d-b54b-4a85-85a4-80b021480939}
   Action aCombineOutputData: Id {e60d4201-2e5a-4e45-91b9-0987642fe282}
   Action aReadInputField1: Id {09026925-47af-4f0d-b345-026e75e997e6}
   Action aReadInputField2: Id {879d4ce2-fa80-469d-ae98-e3a65a92c6ac}
   Action aReadInternalField: Id {d526bcb8-a602-4936-a0ca-348cc77ced31}
   Action aReadNeutralBess: Id {b6f192c3-622c-4489-a181-9ac414869377}
   Action aReadOutputField1: Id {2560e15b-336a-4bdd-a5e9-c733f2196bcb}
   Action aReadOutputField2: Id {23a7dd3d-a6cf-41c7-9f6e-8f42bd580130}
   Action aReadOutputField3: Id {a2de4e77-9600-45d8-8e1d-937b9ee1205f}
   Method ChangeRealEndianess: Id {a4dd5f34-7ca9-4bcb-89f8-7d009941ad52}
   Method MapMeasuringField: Id {51e6d1d3-fcc4-4c41-b2bf-860fdc197c1d}
   Method MapVoltageField: Id {2cec6e0b-54c9-45f5-90b9-49b8eef31073}
   Action ReadDataSFC: Id {d47c650b-b078-4699-aabe-71eb457c26b2}
   Action SFCTipReset: Id {097b2a57-11df-4388-96f3-9b159a6b302d} *)
